// TIA Portal project "Project1" (V16)

(* hardware
DEVICE "S7-1200 station_1"  S7-1200 Station
   slot 0: "Rack_0"  S7-1200 Rack  Rack  V1.0
   slot 1: "PLC_1"  CPU 1214C DC/DC/DC  6ES7 214-1AG40-0XB0  V4.2
   slot 2: "AI 4x13BIT/AQ 2x14BIT_1"  6ES7 234-4HE32-0XB0  V2.1
*)

// ===== PLC "PLC_1"  CPU 1214C DC/DC/DC =====

VAR_GLOBAL   // PLC tag table "Default tag table"
   "Tag_6" AT %MD4 : Real;
   "Tag_9" AT %MW40 : Int;
   "Tag_11" AT %IW64 : Int;
   "Tag_13" AT %Q0.7 : Bool;
   "Tag_10" AT %QW96 : Int;
   "Tag_14" AT %M100.0 : Bool;
   "Tag_8" AT %MW0 : Int;
   "Tag_1" AT %M0.0 : Bool;
END_VAR

ORGANIZATION_BLOCK "Main"   // OB1, LAD, ProgramCycle
TITLE = "Main Program Sweep (Cycle)"
{ S7_Optimized_Access := 'TRUE' }
VERSION : 0.1
   VAR_INPUT
      Initial_Call : Bool;   // Initial call of this OB
      Remanence : Bool;   // =True, if remanent data are available
   END_VAR
BEGIN

REGION Network 1
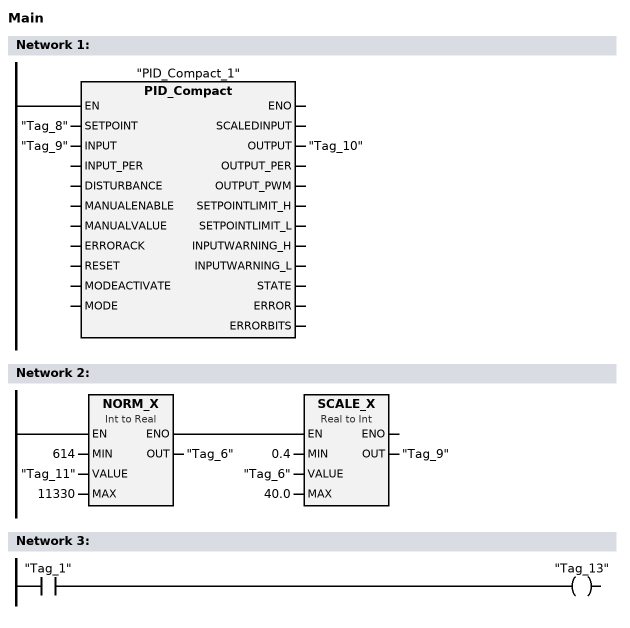
   "PID_Compact_1"(Setpoint := "Tag_8", Input := "Tag_9", Output => "Tag_10");   // PID_Compact
END_REGION

REGION Network 2
   RUNG wire#powerrail
      { S7_Templates := "[SrcType := Int, DestType := Real]" } Normalize(min := 614, value := "Tag_11", max := 11330, out => "Tag_6")
      { S7_Templates := "[SrcType := Real, DestType := Int]" } Scale(min := 0.4, value := "Tag_6", max := 40.0, out => "Tag_9")
   END_RUNG
   // the same network as SCL:
   "Tag_6" := NORM_X(MIN := 614, VALUE := "Tag_11", MAX := 11330);
   "Tag_9" := SCALE_X(MIN := 0.4, VALUE := "Tag_6", MAX := 40.0);
END_REGION

REGION Network 3
   RUNG wire#powerrail
      Contact( "Tag_1" )
      Coil( "Tag_13" )
   END_RUNG
   // the same network as SCL:
   "Tag_13" := "Tag_1";
END_REGION
END_ORGANIZATION_BLOCK